//----------------------------------------------------------------------------//
//            Copyright 2018 Rieckermann Engineering Operations               //
//----------------------------------------------------------------------------//
// Class:       fbDI2                                                         //
// Description:                                                               //
// Normally OFF general alarm single digital input.                           //
//----------------------------------------------------------------------------//
// Revision history:                                                          //
// Rev By               Date        CC        Note                            //
// 2.0 David Paspa      30-Jan-2018 NA        Reboot for S7-1500.             //
// 0.5 Khairul Basar    02-Oct-2009 CC-09/016 NW4 DI changed from NC to NO.   //
// 0.4 Mr. Khoon        01-Oct-2009 CC-09/016 Mode=Initialized,OOS coded.     //
// 0.3 Khairul Basar    30-Sep-2009           Mode=2 initialized and Out of   //
//                                            Service without Alarm.          //
// 0.2 Khairul Basar    31-Aug-2009 CC-09/016 Mode=1 initialized.             //
// 0.1 Khairul Basar    03-Aug-2009           Initial design.                 //
//----------------------------------------------------------------------------//
FUNCTION_BLOCK "fbDI2"
TITLE = DI2 : General alarm single digital input Normally OFF
{ S7_Optimized_Access := 'TRUE' }
NAME : fbDI2
AUTHOR : REO
VERSION : 2.0

//----------------------------------------------------------------------------//
// Declare interface and variables:                                           //
//----------------------------------------------------------------------------//
VAR
    p : "udtDI2";            // Block data interface
END_VAR

VAR DB_SPECIFIC
    b { ExternalAccessible := 'False'; ExternalVisible := 'False'; ExternalWritable := 'False'} : Array[0..15] of Bool;
    w { ExternalAccessible := 'False'; ExternalVisible := 'False'; ExternalWritable := 'False'} AT b : Word;
END_VAR

VAR_TEMP
    tPV : Bool;              // Temporary processed DI signal
END_VAR

BEGIN
NETWORK
TITLE = Process Digital Input Signal
    //------------------------------------------------------------------------//
    // INPUTS   INPUTS   INPUTS   INPUTS   INPUTS   INPUTS   INPUTS   INPUTS  //
    // INPUTS   INPUTS   INPUTS   INPUTS   INPUTS   INPUTS   INPUTS   INPUTS  //
    //                                                                        //
    // Calculate the process value based on input:                            //
    //------------------------------------------------------------------------//
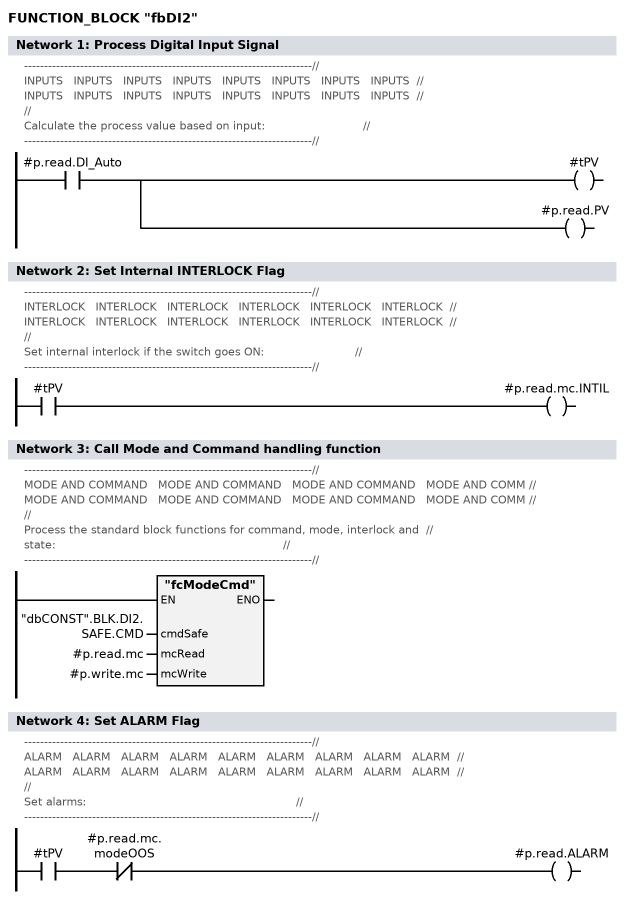
    A #p.read.DI_Auto;
    = #tPV;
    = #p.read.PV;

NETWORK
TITLE = Set Internal INTERLOCK Flag
    //------------------------------------------------------------------------//
    // INTERLOCK   INTERLOCK   INTERLOCK   INTERLOCK   INTERLOCK   INTERLOCK  //
    // INTERLOCK   INTERLOCK   INTERLOCK   INTERLOCK   INTERLOCK   INTERLOCK  //
    //                                                                        //
    // Set internal interlock if the switch goes ON:                          //
    //------------------------------------------------------------------------//
    A #tPV;
    = #p.read.mc.INTIL;

NETWORK
TITLE = Call Mode and Command handling function
    //------------------------------------------------------------------------//
    // MODE AND COMMAND   MODE AND COMMAND   MODE AND COMMAND   MODE AND COMM //
    // MODE AND COMMAND   MODE AND COMMAND   MODE AND COMMAND   MODE AND COMM //
    //                                                                        //
    // Process the standard block functions for command, mode, interlock and  //
    // state:                                                                 //
    //------------------------------------------------------------------------//
    CALL "fcModeCmd"
    (   cmdSafe              := "dbCONST".BLK.DI2.SAFE.CMD ,
        mcRead             := #p.read.mc ,
        mcWrite              := #p.write.mc
    );

NETWORK
TITLE = Set ALARM Flag
    //------------------------------------------------------------------------//
    // ALARM   ALARM   ALARM   ALARM   ALARM   ALARM   ALARM   ALARM   ALARM  //
    // ALARM   ALARM   ALARM   ALARM   ALARM   ALARM   ALARM   ALARM   ALARM  //
    //                                                                        //
    // Set alarms:                                                            //
    //------------------------------------------------------------------------//
    A #tPV;
    AN #p.read.mc.modeOOS;
    = #p.read.ALARM;

NETWORK
TITLE = Set Device State to Enabled if switch is off
    //------------------------------------------------------------------------//
    // STATE   STATE   STATE   STATE   STATE   STATE   STATE   STATE   STATE  //
    // STATE   STATE   STATE   STATE   STATE   STATE   STATE   STATE   STATE  //
    //                                                                        //
    // ENABLED if switch is off:                                              //
    //------------------------------------------------------------------------//
    AN #tPV;
    JCN _a;
    L "dbCONST".BLK.DI2.STATE.ENABLED;
    T #p.read.mc.STATE;
    R #p.read.mc.ERROR;
_a:   NOP 0;

NETWORK
TITLE = Setting Device State to ALARM
    //------------------------------------------------------------------------//
    // ALARM if switch is on and not OOS:                                     //
    //------------------------------------------------------------------------//
    A #tPV;
    AN #p.read.mc.modeOOS;
    JCN _b;
    L "dbCONST".BLK.DI2.STATE.ALARM;
    T #p.read.mc.STATE;
    S #p.read.mc.ERROR;
_b:   NOP 0;

NETWORK
TITLE = Pack the alarm bit
    //------------------------------------------------------------------------//
    // Pack the alarm bit into an integer for the HMI to read:                //
    // Alarms are arranged in the following Little Endian order...            //
    // Word   1                                0                              //
    // Bit    0   1   2   3   4   5   6   7    8   9  10  11  12  13  14  15  //
    // Order  9  10  11  12  13  14  15  16    1   2   3   4   5   6   7   8  //
    //------------------------------------------------------------------------//
    A #p.read.ALARM;
    = #b[8];
    L #w;
    T #p.read.mc.ALARM;

END_FUNCTION_BLOCK
